(* CODESYS project StopLights_TONonly.project

Project tree, tasks and I/O mapping:
  Device : CODESYS Control Win V3, 3S - Smart Software Solutions GmbH, order no. 305021, version 3.5.11.40
    application Application
      libraries: Standard, * (System)
      task MainTask (cyclic, interval t#20ms, priority 1) calls PLC_PRG
      task VISU_TASK (cyclic, interval 100 ms, priority 31) calls VisuElems.Visu_Prg
      program PLC_PRG [LD]
      visualisation Visualization
  global variables GVL
  text list GlobalTextList
*)

// GVL
{attribute 'qualified_only'}
VAR_GLOBAL
END_VAR

// Device/Application/PLC_PRG
PROGRAM PLC_PRG
VAR
	start: BOOL;
	stop: BOOL;
	// Holding bit
	H: BOOL;
	//Green Light
	Green: BOOL;
	//Yellow light
	Yellow: BOOL;
	//Red light
	Red: BOOL;
	//TON 0,1,2,3 timers
	TON_0: TON;
	TON_1: TON;
	TON_2: TON;
	TON_3: TON;
	// Dummy 1, 2, 3 bit: main use to see output is working
	db: BOOL;
	db2: BOOL;
	db3: BOOL;
	// Delays yellow light by 1 second interval
	Timer_delayer: TON;
	// Delays yellow light by 1 second interval
	Timer_delayer_2: TON;
END_VAR

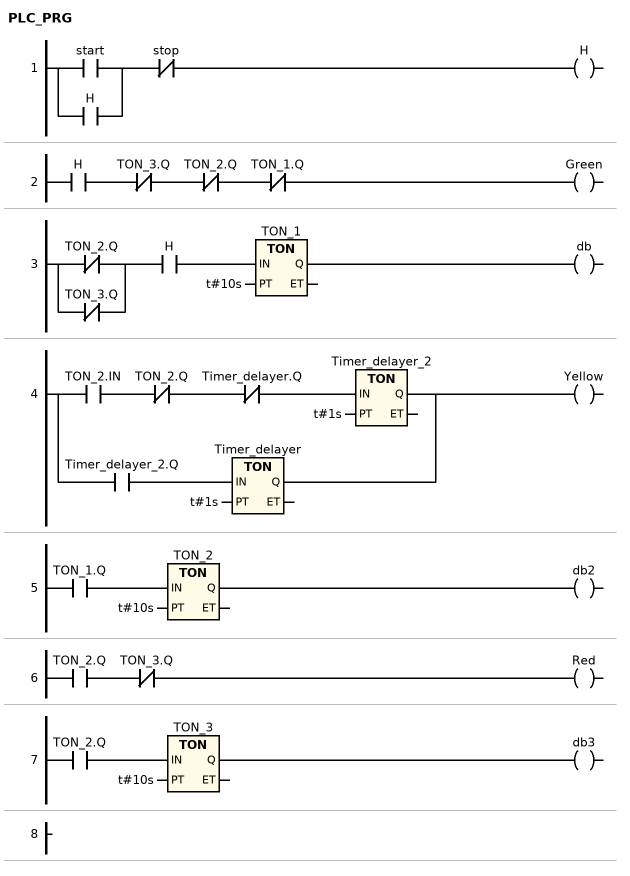
// NETWORK 1
H := (start OR H) AND NOT stop;

// NETWORK 2
Green := H AND NOT TON_3.Q AND NOT TON_2.Q AND NOT TON_1.Q;

// NETWORK 3
TON_1(IN := (NOT TON_2.Q OR NOT TON_3.Q) AND H, PT := t#10s); // TON
db := TON_1.Q;

// NETWORK 4
Timer_delayer_2(IN := TON_2.IN AND NOT TON_2.Q AND NOT Timer_delayer.Q, PT := t#1s); // TON
Timer_delayer(IN := Timer_delayer_2.Q, PT := t#1s); // TON
Yellow := Timer_delayer_2.Q OR Timer_delayer.Q;

// NETWORK 5
TON_2(IN := TON_1.Q, PT := t#10s); // TON
db2 := TON_2.Q;

// NETWORK 6
Red := TON_2.Q AND NOT TON_3.Q;

// NETWORK 7
TON_3(IN := TON_2.Q, PT := t#10s); // TON
db3 := TON_3.Q;

// NETWORK 8

END_PROGRAM

// Device/Application/Visualization
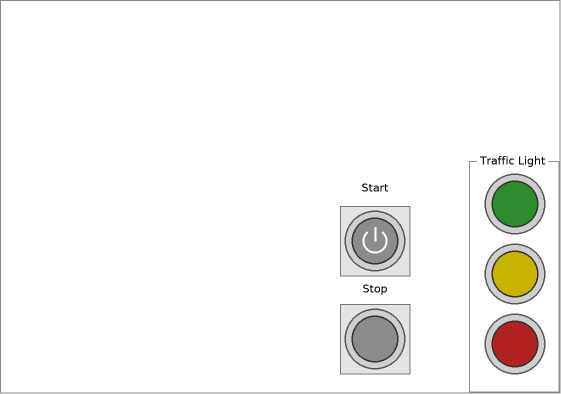
VISUALIZATION Visualization  // 561x394
    Lamp1 (480,169 70x70), variable: PLC_PRG.Green, style: Lamp-Lamp1-Green
    Lamp1 (480,239 70x70), variable: PLC_PRG.Yellow, style: Lamp-Lamp1-Yellow
    Lamp1 (480,309 70x70), variable: PLC_PRG.Red, style: Lamp-Lamp1-Red
    PowerSwitch (340,206 70x70), variable: PLC_PRG.start, behaviour: TAP, style: Switch-PowerSwitch-Gray
    PushSwitch (340,304 70x70), variable: PLC_PRG.stop, behaviour: TAP, style: Switch-PushSwitch-Gray
    Label (300,173 150x30), "Start"
    Label (300,274 150x30), "Stop"
    GroupBox (469,153 90x239), "Traffic Light"
END_VISUALIZATION
